(* Logix 5000 project; controller cal1615 1756-L62 rev 20.19; software revision 20.05; part 52 of 82 *)
(* tags used below, declared in another part *)
   FAULT : BOOL;   // Fault AFI
   HMI : BOOL;   // AFI HMI
   p01r09_pb_global_reset : BOOL;   // System Modes PB: Global Fault Reset
   p02_real_from_hmi : hmi_real;   // MOP HMI Iface Real from HMI
   p23_ai_lfl : REAL;   // Impreg Inputs LFL level
   p23_ai_metering_roll_amps : REAL;   // Impreg Analog Input Impreg Metering Roll Motor Current
   p23_ai_metering_roll_hz : REAL;   // Impreg Analog Input Impreg Metering Roll Motor Max Hz
   p23_ai_metering_roll_speed_fpm : REAL;   // Impreg Analog Input Impreg Roll Speed
   p23_ai_prs : REAL;   // Impreg Analog Inputs Impreg Enclosure Pressure
   p23_ai_servo_ds_position : REAL;   // Impreg Servo Drive Side Actual Position
   p23_ai_servo_ds_torque : REAL;   // Impreg Servo Drive Side Actual Torque
   p23_ai_servo_os_position : REAL;   // Impreg Inputs Servo Operator Side Position
   p23_ai_servo_os_torque : REAL;   // Impreg Inputs Servo Operator Side Torque
   p23_ai_servo_os_velocity : REAL;   // Impreg Inputs Servo Operator Side Velocity
   p23_ai_supply_amps : REAL;   // Impreg Analog Inputs Supply Fan VFD Amps
   p23_ai_supply_hz : REAL;   // Impreg Analog Inputs Supply Fan VFD Hz
   p23_ai_supply_rpm : REAL;   // Impreg Analog Inputs Supply Fan RPM
   p23_di_spring : acs800_di_normal;
   p23_di_supply : acs800_di_normal;   // Impreg Supply VFD VFD Inputs
   p23_dint_to_hmi : DINT[17];   // Impreg Dint to HMI
   p23_param_lfl_hhl : REAL;   // Impreg Parameter LFL High High Limit
   p23_param_lfl_hl : REAL;   // Impreg Parameters LFL High Limit
   p23_param_zone_pressure : REAL;   // MOP HMI Iface Parameters Minimum Pressure
   p23_real_to_hmi : REAL[112];   // Impreg Real to HMI
   p23_servo_os_warning : SYS_ENC_WITH_ZERO_BIT;   // Impreg Dint to HMI Servo Operator Side Warning
   p23r01 : routine;   // Impreg Main
   p23r02 : routine;   // Impreg Misc Control
   p23r05 : routine;   // Impreg Dint to HMI
   p23r05_supply_status : DINT;
   p23r05_timer_fault : TIMER[4];   // Impreg Dint to HMI Timer Fault
   p23r05_timer_warning : TIMER[4];   // Impreg Dint to HMI Timer Warning
   p23r06 : routine;   // Impreg Real to HMI
   p23r06_timer_fault : TIMER[4];   // Impreg Real to HMI Fault Delay
   p23r06_timer_warning : TIMER[4];   // Impreg Real to HMI Warning Delay
   p23r07 : routine;   // Impreg Alarms
   p23r07_timer_fault : TIMER[4];   // Impreg Alarms Fault Delay
   p23r07_timer_warning : TIMER[4];   // Impreg Alarms Warning Delay
   p23r11 : routine;   // Impreg Servo Operator Side
   p23r11_pos_offset : REAL;
   p23r12 : routine;   // Impreg Servo Drive Side
   p23r12_pos_offset : REAL;
   p23r13 : routine;
   p23r13_vfd_stopped : BOOL;   // Impreg Supply VFD Stopped
   p23r15 : routine;   // Impreg Metering Roll VFD
   p32r13_request_auto_stop : BOOL;   // Impreg Supply VFD Request Auto Stop
(* P23_Impreg, continued *)

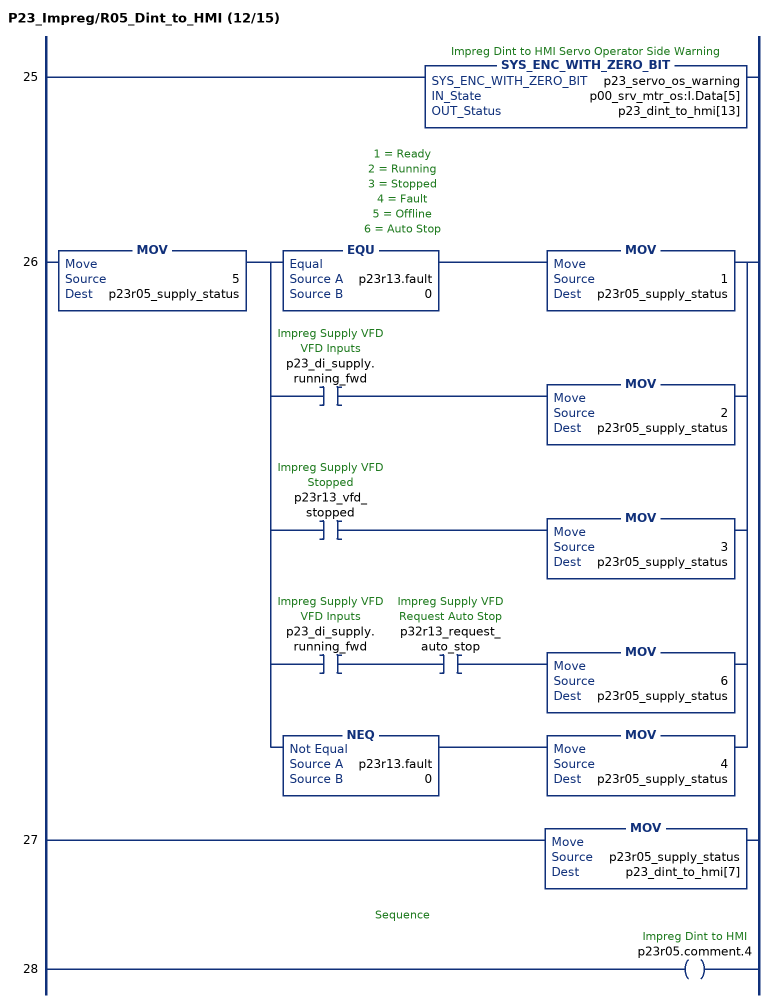
   [picture p1017: P23_Impreg/R05_Dint_to_HMI rungs 25-28]
   25: SYS_ENC_WITH_ZERO_BIT(p23_servo_os_warning,p00_srv_mtr_os:I.Data[5],p23_dint_to_hmi[13]);
   // 1 = Ready
   // 2 = Running
   // 3 = Stopped
   // 4 = Fault
   // 5 = Offline
   // 6 = Auto Stop
   26: MOV(5,p23r05_supply_status)[EQU(p23r13.fault,0) MOV(1,p23r05_supply_status) ,XIC(p23_di_supply.running_fwd) MOV(2,p23r05_supply_status) ,XIC(p23r13_vfd_stopped) MOV(3,p23r05_supply_status) ,XIC(p23_di_supply.running_fwd) XIC(p32r13_request_auto_stop) MOV(6,p23r05_supply_status) ,NEQ(p23r13.fault,0) MOV(4,p23r05_supply_status) ];
   27: MOV(p23r05_supply_status,p23_dint_to_hmi[7]);
   // Sequence
   28: OTE(p23r05.comment.4);
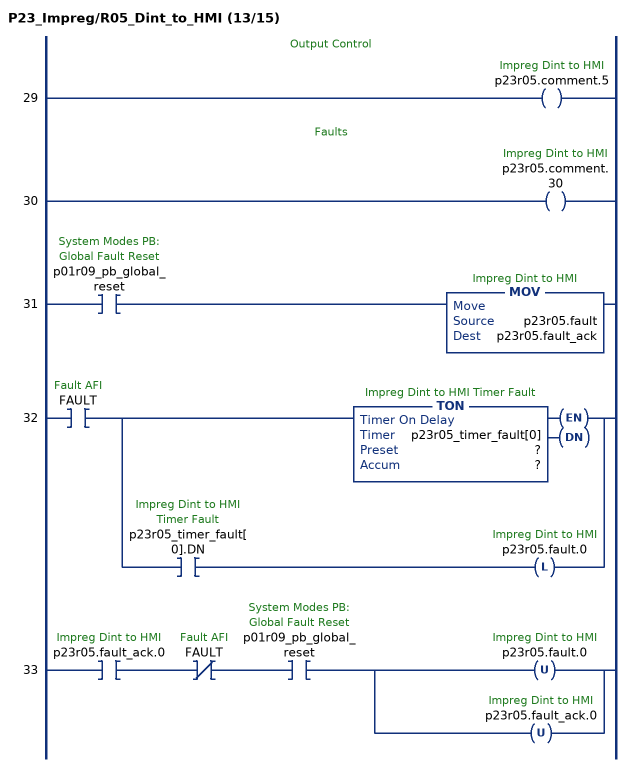
   // Output Control
   29: OTE(p23r05.comment.5);
   // Faults
   30: OTE(p23r05.comment.30);
   31: XIC(p01r09_pb_global_reset)MOV(p23r05.fault,p23r05.fault_ack);
   32: XIC(FAULT)[TON(p23r05_timer_fault[0],?,?) ,XIC(p23r05_timer_fault[0].DN) OTL(p23r05.fault.0) ];
   33: XIC(p23r05.fault_ack.0)XIO(FAULT)XIC(p01r09_pb_global_reset)[OTU(p23r05.fault.0) ,OTU(p23r05.fault_ack.0) ];
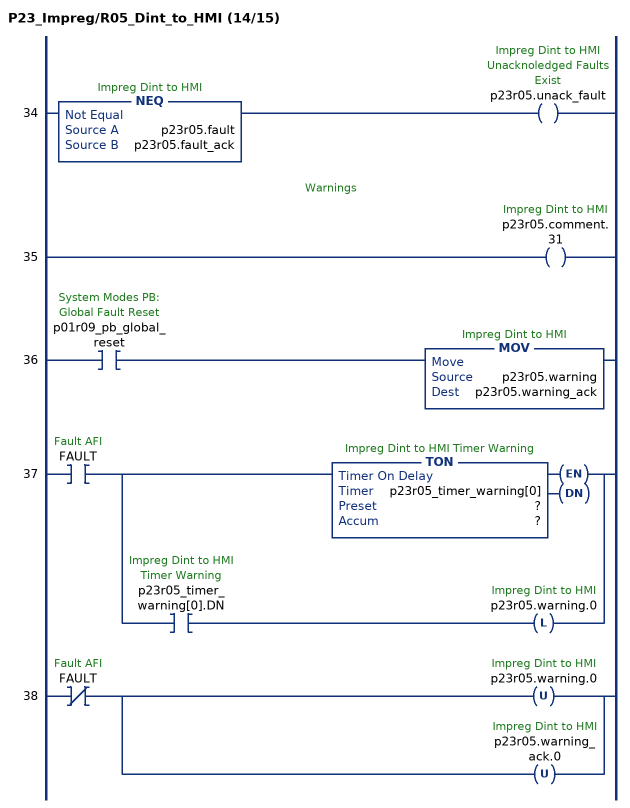
   34: NEQ(p23r05.fault,p23r05.fault_ack)OTE(p23r05.unack_fault);
   // Warnings
   35: OTE(p23r05.comment.31);
   36: XIC(p01r09_pb_global_reset)MOV(p23r05.warning,p23r05.warning_ack);
   37: XIC(FAULT)[TON(p23r05_timer_warning[0],?,?) ,XIC(p23r05_timer_warning[0].DN) OTL(p23r05.warning.0) ];
   38: XIO(FAULT)[OTU(p23r05.warning.0) ,OTU(p23r05.warning_ack.0) ];
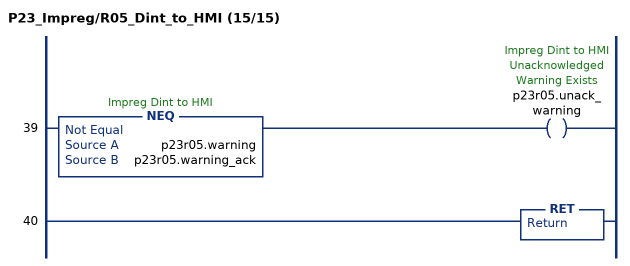
   39: NEQ(p23r05.warning,p23r05.warning_ack)OTE(p23r05.unack_warning);
   40: RET();
END_ROUTINE

ROUTINE R06_Real_to_HMI   (* ladder *)
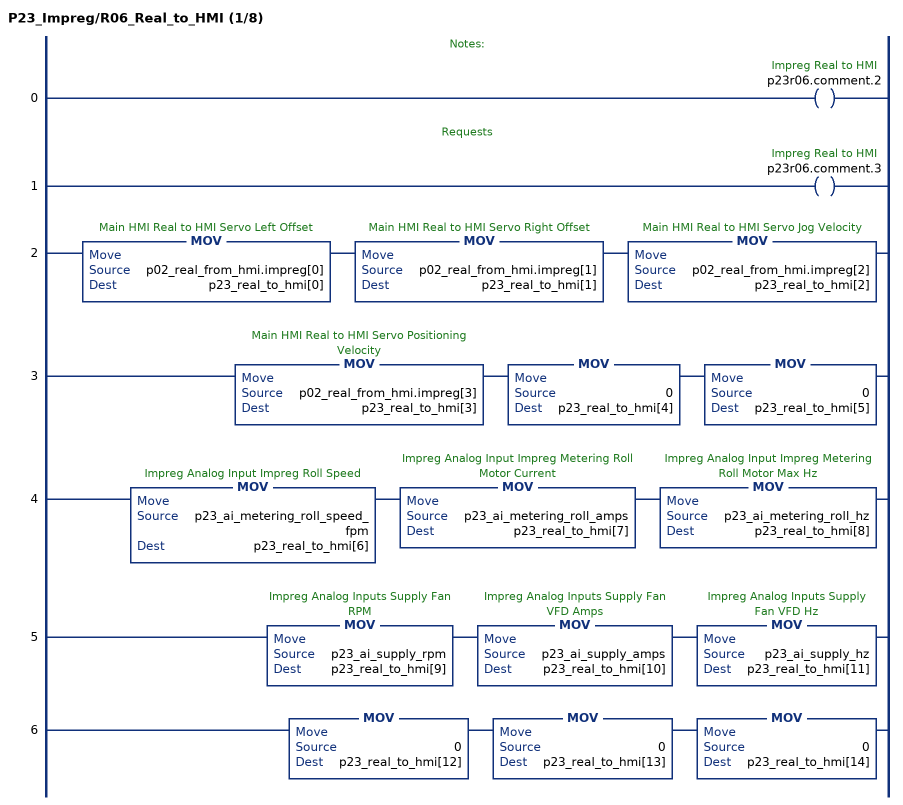
   // Notes:
   0: OTE(p23r06.comment.2);
   // Requests
   1: OTE(p23r06.comment.3);
   2: MOV(p02_real_from_hmi.impreg[0],p23_real_to_hmi[0])MOV(p02_real_from_hmi.impreg[1],p23_real_to_hmi[1])MOV(p02_real_from_hmi.impreg[2],p23_real_to_hmi[2]);
   3: MOV(p02_real_from_hmi.impreg[3],p23_real_to_hmi[3])MOV(0,p23_real_to_hmi[4])MOV(0,p23_real_to_hmi[5]);
   4: MOV(p23_ai_metering_roll_speed_fpm,p23_real_to_hmi[6])MOV(p23_ai_metering_roll_amps,p23_real_to_hmi[7])MOV(p23_ai_metering_roll_hz,p23_real_to_hmi[8]);
   5: MOV(p23_ai_supply_rpm,p23_real_to_hmi[9])MOV(p23_ai_supply_amps,p23_real_to_hmi[10])MOV(p23_ai_supply_hz,p23_real_to_hmi[11]);
   6: MOV(0,p23_real_to_hmi[12])MOV(0,p23_real_to_hmi[13])MOV(0,p23_real_to_hmi[14]);
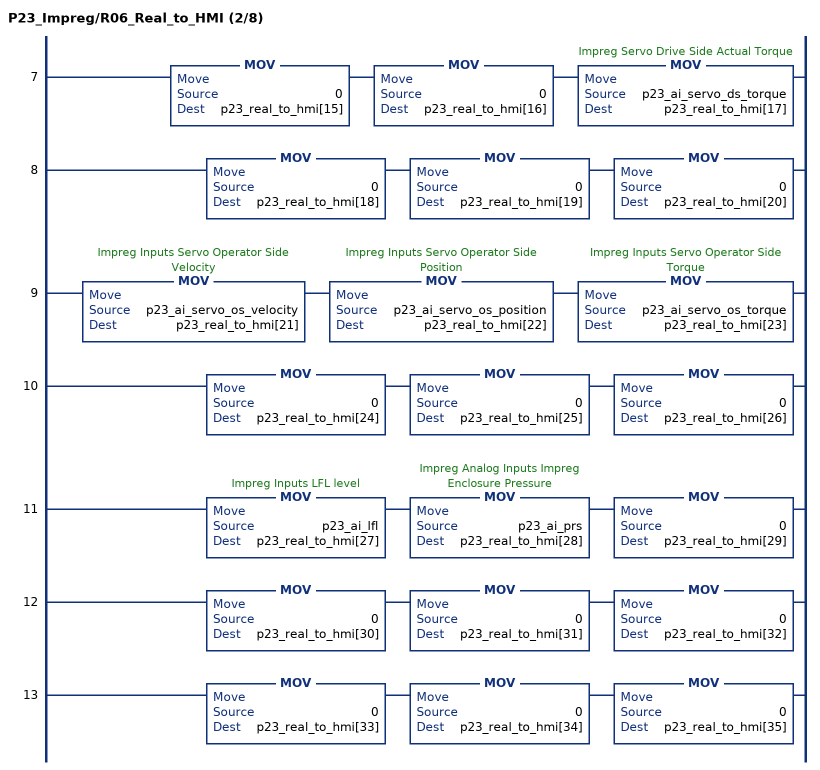
   7: MOV(0,p23_real_to_hmi[15])MOV(0,p23_real_to_hmi[16])MOV(p23_ai_servo_ds_torque,p23_real_to_hmi[17]);
   8: MOV(0,p23_real_to_hmi[18])MOV(0,p23_real_to_hmi[19])MOV(0,p23_real_to_hmi[20]);
   9: MOV(p23_ai_servo_os_velocity,p23_real_to_hmi[21])MOV(p23_ai_servo_os_position,p23_real_to_hmi[22])MOV(p23_ai_servo_os_torque,p23_real_to_hmi[23]);
   10: MOV(0,p23_real_to_hmi[24])MOV(0,p23_real_to_hmi[25])MOV(0,p23_real_to_hmi[26]);
   11: MOV(p23_ai_lfl,p23_real_to_hmi[27])MOV(p23_ai_prs,p23_real_to_hmi[28])MOV(0,p23_real_to_hmi[29]);
   12: MOV(0,p23_real_to_hmi[30])MOV(0,p23_real_to_hmi[31])MOV(0,p23_real_to_hmi[32]);
   13: MOV(0,p23_real_to_hmi[33])MOV(0,p23_real_to_hmi[34])MOV(0,p23_real_to_hmi[35]);
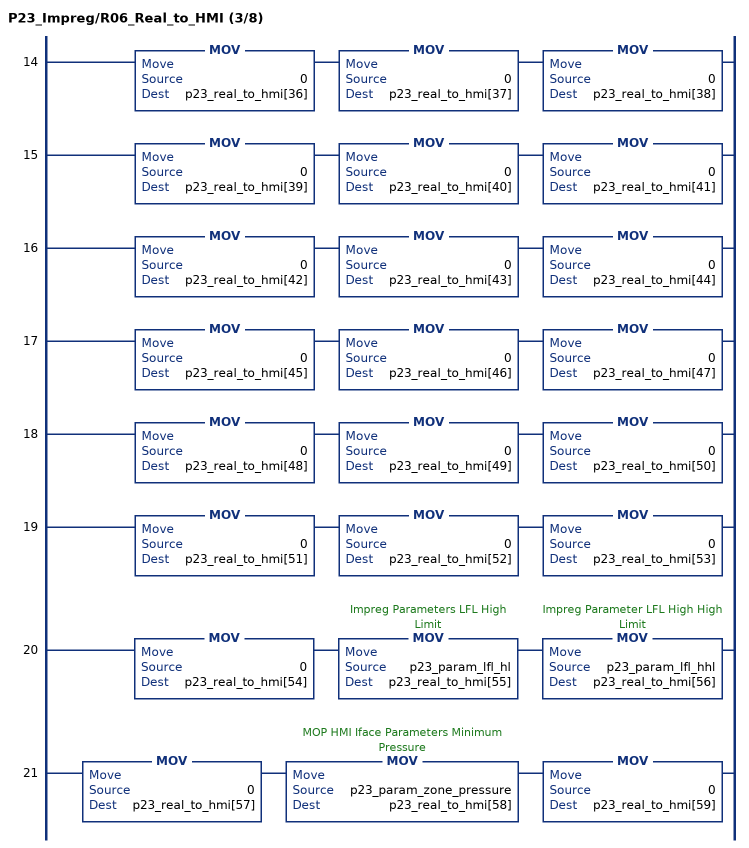
   14: MOV(0,p23_real_to_hmi[36])MOV(0,p23_real_to_hmi[37])MOV(0,p23_real_to_hmi[38]);
   15: MOV(0,p23_real_to_hmi[39])MOV(0,p23_real_to_hmi[40])MOV(0,p23_real_to_hmi[41]);
   16: MOV(0,p23_real_to_hmi[42])MOV(0,p23_real_to_hmi[43])MOV(0,p23_real_to_hmi[44]);
   17: MOV(0,p23_real_to_hmi[45])MOV(0,p23_real_to_hmi[46])MOV(0,p23_real_to_hmi[47]);
   18: MOV(0,p23_real_to_hmi[48])MOV(0,p23_real_to_hmi[49])MOV(0,p23_real_to_hmi[50]);
   19: MOV(0,p23_real_to_hmi[51])MOV(0,p23_real_to_hmi[52])MOV(0,p23_real_to_hmi[53]);
   20: MOV(0,p23_real_to_hmi[54])MOV(p23_param_lfl_hl,p23_real_to_hmi[55])MOV(p23_param_lfl_hhl,p23_real_to_hmi[56]);
   21: MOV(0,p23_real_to_hmi[57])MOV(p23_param_zone_pressure,p23_real_to_hmi[58])MOV(0,p23_real_to_hmi[59]);
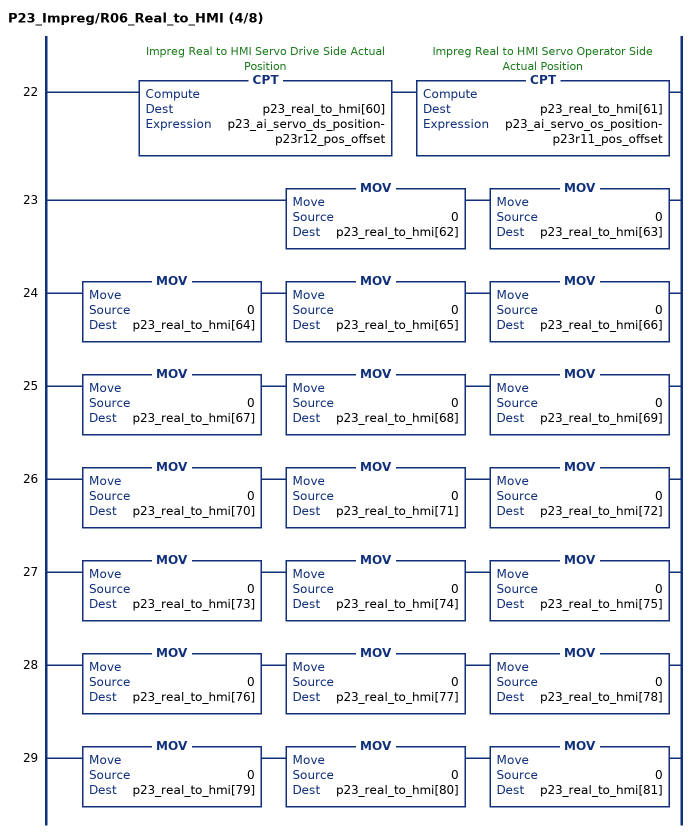
   22: CPT(p23_real_to_hmi[60],p23_ai_servo_ds_position-p23r12_pos_offset)CPT(p23_real_to_hmi[61],p23_ai_servo_os_position-p23r11_pos_offset);
   23: MOV(0,p23_real_to_hmi[62])MOV(0,p23_real_to_hmi[63]);
   24: MOV(0,p23_real_to_hmi[64])MOV(0,p23_real_to_hmi[65])MOV(0,p23_real_to_hmi[66]);
   25: MOV(0,p23_real_to_hmi[67])MOV(0,p23_real_to_hmi[68])MOV(0,p23_real_to_hmi[69]);
   26: MOV(0,p23_real_to_hmi[70])MOV(0,p23_real_to_hmi[71])MOV(0,p23_real_to_hmi[72]);
   27: MOV(0,p23_real_to_hmi[73])MOV(0,p23_real_to_hmi[74])MOV(0,p23_real_to_hmi[75]);
   28: MOV(0,p23_real_to_hmi[76])MOV(0,p23_real_to_hmi[77])MOV(0,p23_real_to_hmi[78]);
   29: MOV(0,p23_real_to_hmi[79])MOV(0,p23_real_to_hmi[80])MOV(0,p23_real_to_hmi[81]);
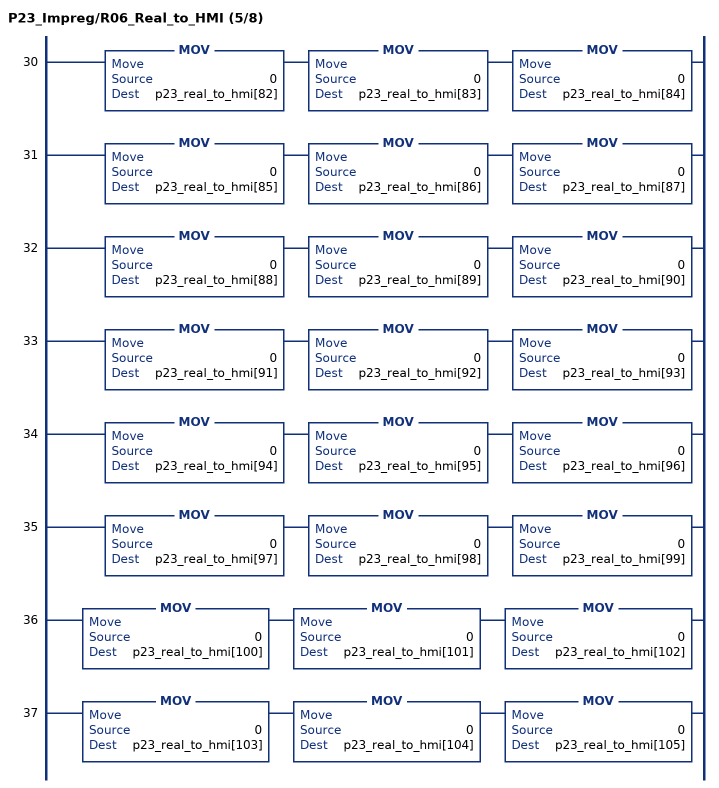
   30: MOV(0,p23_real_to_hmi[82])MOV(0,p23_real_to_hmi[83])MOV(0,p23_real_to_hmi[84]);
   31: MOV(0,p23_real_to_hmi[85])MOV(0,p23_real_to_hmi[86])MOV(0,p23_real_to_hmi[87]);
   32: MOV(0,p23_real_to_hmi[88])MOV(0,p23_real_to_hmi[89])MOV(0,p23_real_to_hmi[90]);
   33: MOV(0,p23_real_to_hmi[91])MOV(0,p23_real_to_hmi[92])MOV(0,p23_real_to_hmi[93]);
   34: MOV(0,p23_real_to_hmi[94])MOV(0,p23_real_to_hmi[95])MOV(0,p23_real_to_hmi[96]);
   35: MOV(0,p23_real_to_hmi[97])MOV(0,p23_real_to_hmi[98])MOV(0,p23_real_to_hmi[99]);
   36: MOV(0,p23_real_to_hmi[100])MOV(0,p23_real_to_hmi[101])MOV(0,p23_real_to_hmi[102]);
   37: MOV(0,p23_real_to_hmi[103])MOV(0,p23_real_to_hmi[104])MOV(0,p23_real_to_hmi[105]);
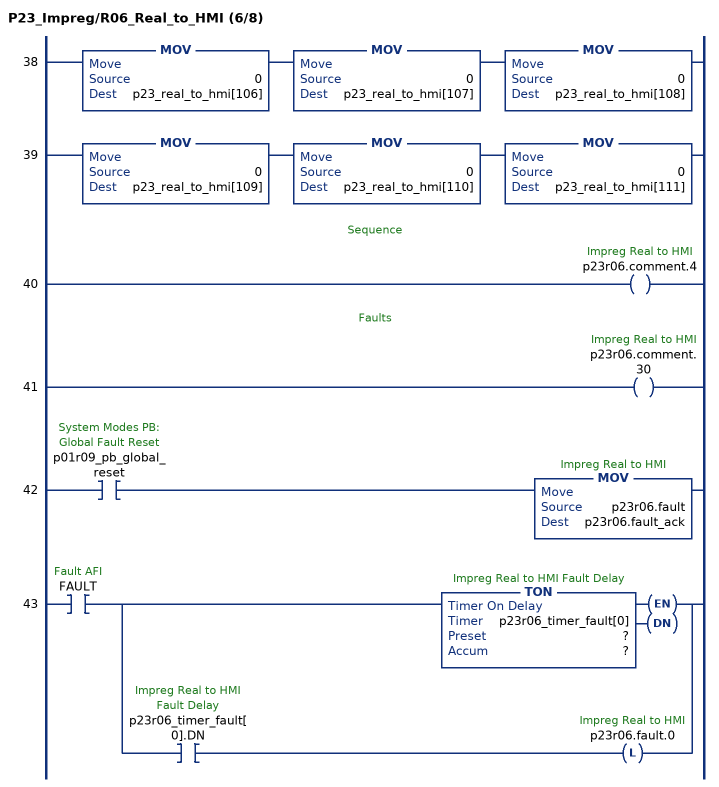
   38: MOV(0,p23_real_to_hmi[106])MOV(0,p23_real_to_hmi[107])MOV(0,p23_real_to_hmi[108]);
   39: MOV(0,p23_real_to_hmi[109])MOV(0,p23_real_to_hmi[110])MOV(0,p23_real_to_hmi[111]);
   // Sequence
   40: OTE(p23r06.comment.4);
   // Faults
   41: OTE(p23r06.comment.30);
   42: XIC(p01r09_pb_global_reset)MOV(p23r06.fault,p23r06.fault_ack);
   43: XIC(FAULT)[TON(p23r06_timer_fault[0],?,?) ,XIC(p23r06_timer_fault[0].DN) OTL(p23r06.fault.0) ];
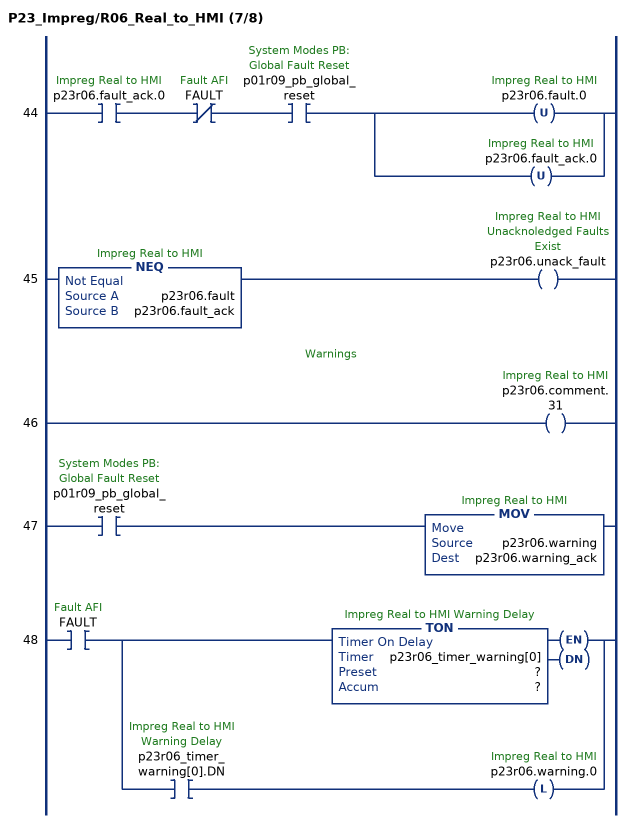
   44: XIC(p23r06.fault_ack.0)XIO(FAULT)XIC(p01r09_pb_global_reset)[OTU(p23r06.fault.0) ,OTU(p23r06.fault_ack.0) ];
   45: NEQ(p23r06.fault,p23r06.fault_ack)OTE(p23r06.unack_fault);
   // Warnings
   46: OTE(p23r06.comment.31);
   47: XIC(p01r09_pb_global_reset)MOV(p23r06.warning,p23r06.warning_ack);
   48: XIC(FAULT)[TON(p23r06_timer_warning[0],?,?) ,XIC(p23r06_timer_warning[0].DN) OTL(p23r06.warning.0) ];
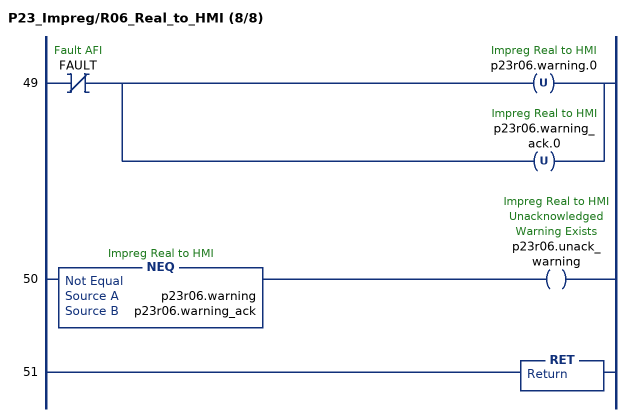
   49: XIO(FAULT)[OTU(p23r06.warning.0) ,OTU(p23r06.warning_ack.0) ];
   50: NEQ(p23r06.warning,p23r06.warning_ack)OTE(p23r06.unack_warning);
   51: RET();
END_ROUTINE

ROUTINE R07_Alarms   (* ladder *)
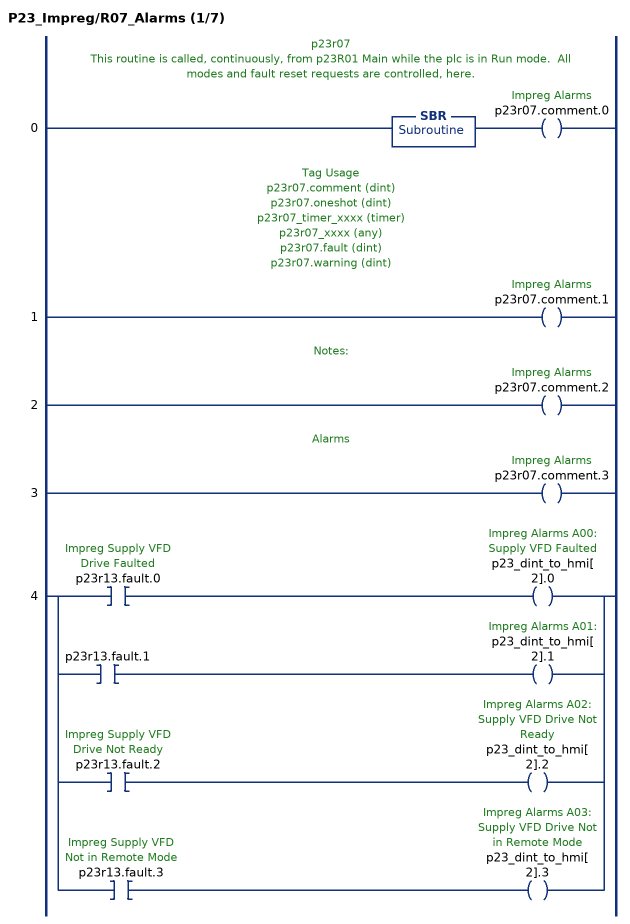
   // p23r07
   // This routine is called, continuously, from p23R01 Main while the plc is in Run mode.  All modes and fault reset requests are controlled, here.
   0: SBR()OTE(p23r07.comment.0);
   // Tag Usage
   // p23r07.comment (dint)
   // p23r07.oneshot (dint)
   // p23r07_timer_xxxx (timer)
   // p23r07_xxxx (any)
   // p23r07.fault (dint)
   // p23r07.warning (dint)
   1: OTE(p23r07.comment.1);
   // Notes:
   2: OTE(p23r07.comment.2);
   // Alarms
   3: OTE(p23r07.comment.3);
   4: [XIC(p23r13.fault.0) OTE(p23_dint_to_hmi[2].0) ,XIC(p23r13.fault.1) OTE(p23_dint_to_hmi[2].1) ,XIC(p23r13.fault.2) OTE(p23_dint_to_hmi[2].2) ,XIC(p23r13.fault.3) OTE(p23_dint_to_hmi[2].3) ];
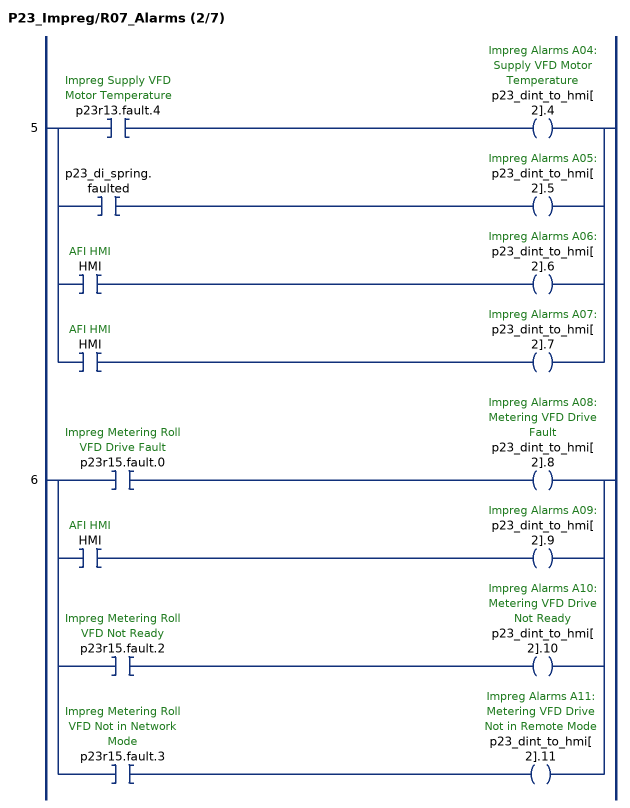
   5: [XIC(p23r13.fault.4) OTE(p23_dint_to_hmi[2].4) ,XIC(p23_di_spring.faulted) OTE(p23_dint_to_hmi[2].5) ,XIC(HMI) OTE(p23_dint_to_hmi[2].6) ,XIC(HMI) OTE(p23_dint_to_hmi[2].7) ];
   6: [XIC(p23r15.fault.0) OTE(p23_dint_to_hmi[2].8) ,XIC(HMI) OTE(p23_dint_to_hmi[2].9) ,XIC(p23r15.fault.2) OTE(p23_dint_to_hmi[2].10) ,XIC(p23r15.fault.3) OTE(p23_dint_to_hmi[2].11) ];
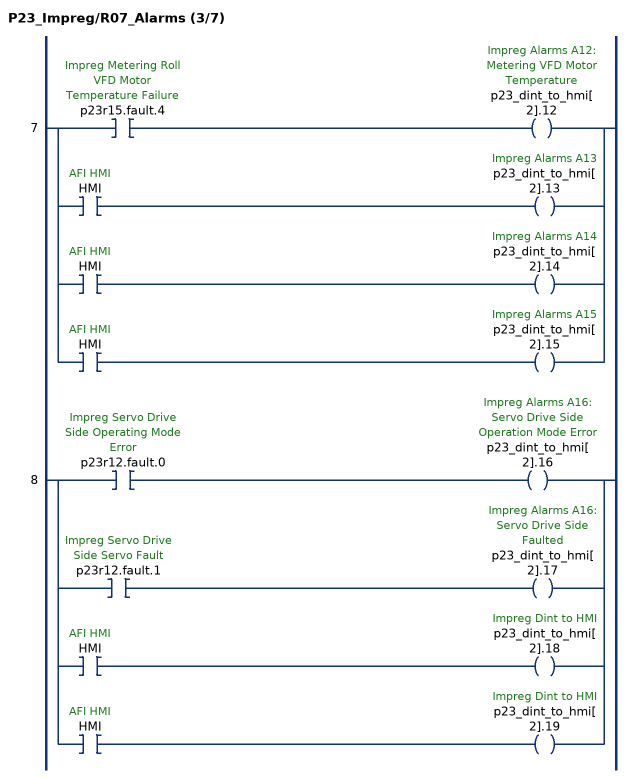
   7: [XIC(p23r15.fault.4) OTE(p23_dint_to_hmi[2].12) ,XIC(HMI) OTE(p23_dint_to_hmi[2].13) ,XIC(HMI) OTE(p23_dint_to_hmi[2].14) ,XIC(HMI) OTE(p23_dint_to_hmi[2].15) ];
   8: [XIC(p23r12.fault.0) OTE(p23_dint_to_hmi[2].16) ,XIC(p23r12.fault.1) OTE(p23_dint_to_hmi[2].17) ,XIC(HMI) OTE(p23_dint_to_hmi[2].18) ,XIC(HMI) OTE(p23_dint_to_hmi[2].19) ];
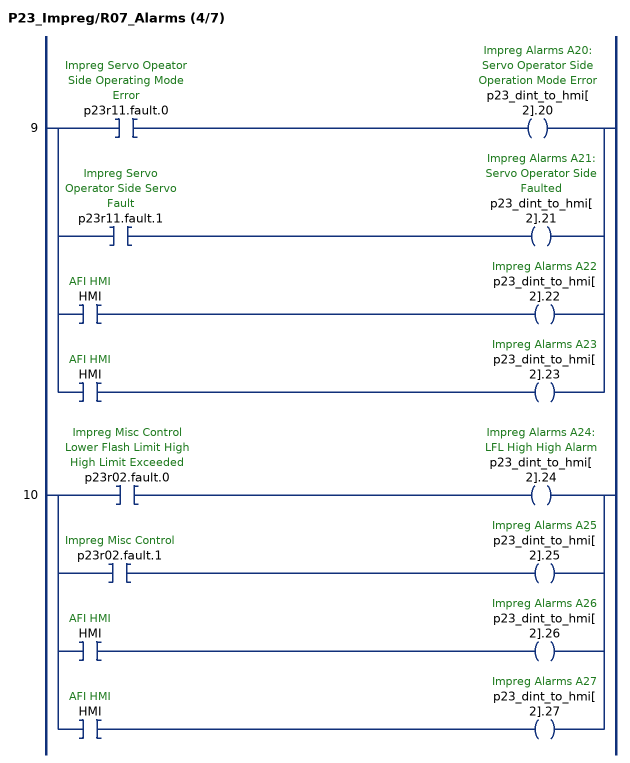
   9: [XIC(p23r11.fault.0) OTE(p23_dint_to_hmi[2].20) ,XIC(p23r11.fault.1) OTE(p23_dint_to_hmi[2].21) ,XIC(HMI) OTE(p23_dint_to_hmi[2].22) ,XIC(HMI) OTE(p23_dint_to_hmi[2].23) ];
   10: [XIC(p23r02.fault.0) OTE(p23_dint_to_hmi[2].24) ,XIC(p23r02.fault.1) OTE(p23_dint_to_hmi[2].25) ,XIC(HMI) OTE(p23_dint_to_hmi[2].26) ,XIC(HMI) OTE(p23_dint_to_hmi[2].27) ];
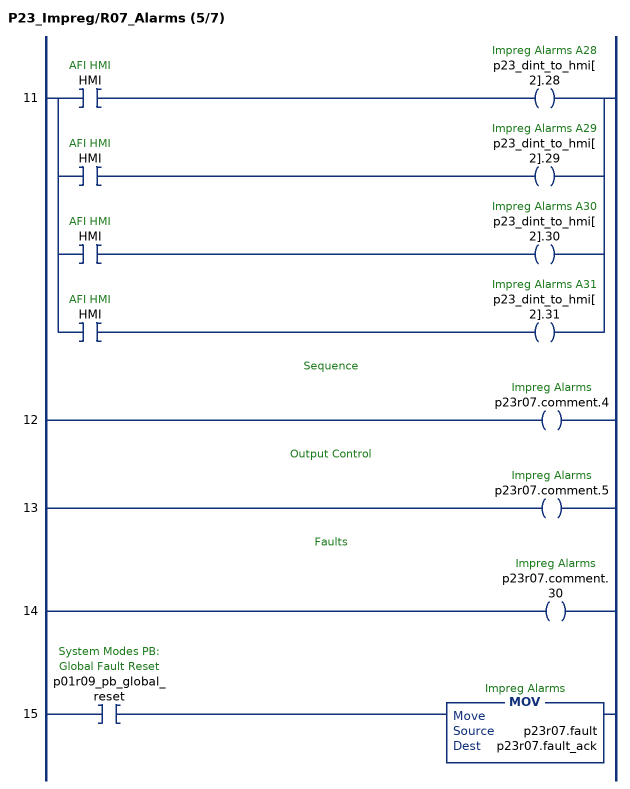
   11: [XIC(HMI) OTE(p23_dint_to_hmi[2].28) ,XIC(HMI) OTE(p23_dint_to_hmi[2].29) ,XIC(HMI) OTE(p23_dint_to_hmi[2].30) ,XIC(HMI) OTE(p23_dint_to_hmi[2].31) ];
   // Sequence
   12: OTE(p23r07.comment.4);
   // Output Control
   13: OTE(p23r07.comment.5);
   // Faults
   14: OTE(p23r07.comment.30);
   15: XIC(p01r09_pb_global_reset)MOV(p23r07.fault,p23r07.fault_ack);
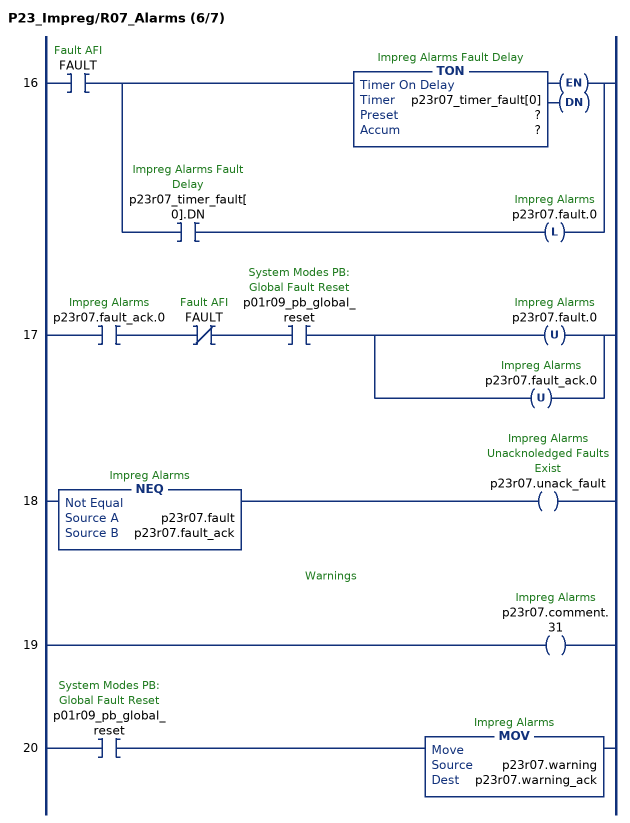
   16: XIC(FAULT)[TON(p23r07_timer_fault[0],?,?) ,XIC(p23r07_timer_fault[0].DN) OTL(p23r07.fault.0) ];
   17: XIC(p23r07.fault_ack.0)XIO(FAULT)XIC(p01r09_pb_global_reset)[OTU(p23r07.fault.0) ,OTU(p23r07.fault_ack.0) ];
   18: NEQ(p23r07.fault,p23r07.fault_ack)OTE(p23r07.unack_fault);
   // Warnings
   19: OTE(p23r07.comment.31);
   20: XIC(p01r09_pb_global_reset)MOV(p23r07.warning,p23r07.warning_ack);
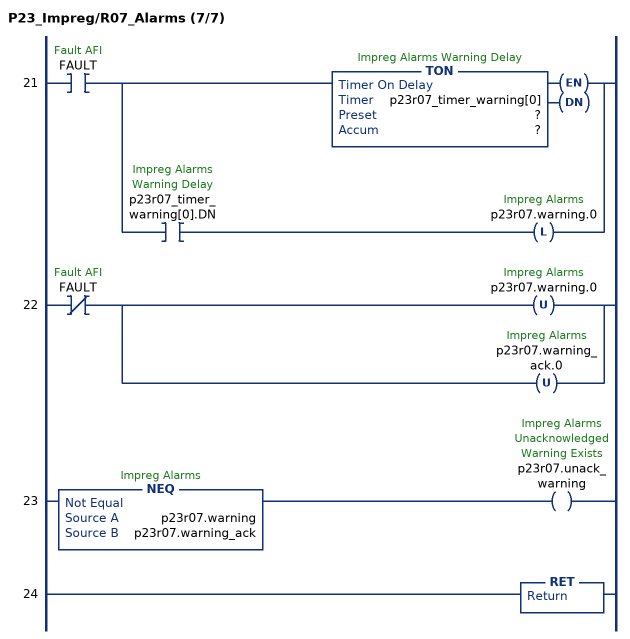
   21: XIC(FAULT)[TON(p23r07_timer_warning[0],?,?) ,XIC(p23r07_timer_warning[0].DN) OTL(p23r07.warning.0) ];
   22: XIO(FAULT)[OTU(p23r07.warning.0) ,OTU(p23r07.warning_ack.0) ];
   23: NEQ(p23r07.warning,p23r07.warning_ack)OTE(p23r07.unack_warning);
   24: RET();
END_ROUTINE
